{attribute 'GeneratedUsingTerminal: EL5001-0011-0016'}
{attribute addProperty BoxType "EL5001-0011-0016"}
{attribute addProperty Description "EL5001-0011 1Ch. SSI Monitor"}
{attribute addProperty Physics "KK"}
{attribute addProperty Id "SSI_InputsAT %I*SSI_Inputs_3B70A31110WcStateAT %I*WcState_9091E0EB2InfoDataAT %I*InfoData_BEF6B88E18"}
{attribute addProperty CRC "3870212281"}
{attribute addProperty Size "30"}
TYPE EL5001_E6AEC0B9 EXTENDS EtcSlaveTerminalBase_947E5A46 :
STRUCT
	{attribute addProperty Name "SSI_Inputs"}
	SSI_Inputs : SSI_Inputs_3B70A311;
	{attribute addProperty Name "WcState"}
	WcState : WcState_9091E0EB;
	{attribute addProperty Name "InfoData"}
	InfoData : InfoData_BEF6B88E;
END_STRUCT
END_TYPE

(* stored: Version 1.2.0.0, ProductVersion 3.1.4024.11
   DUT EL5001_E6AEC0B9: Id {6484441e-667a-4b37-9c0d-0730fc2d9b4f} *)
